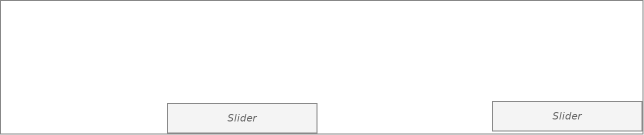
VISUALIZATION Visualization  // 644x135
    Slider (167,103 150x30), variable: MAIN.r_Tao, scale 0..10
    Slider (492,101 150x30), variable: MAIN.r_Input, scale 0..100
END_VISUALIZATION

(* stored: Version 1.1.0.1, ProductVersion 3.1.4022.12
   Visu Visualization: Id {2c0a86d7-c444-4b64-8f00-f546e31c53b7} *)
